# EPICS substitutions: citestApp/Db/user.substitutions
# Example substitutions file

file "db/dbExample1.db" {
    { user = "sdcswd" }
}

file db/dbExample2.db {
    pattern { user, no, scan }
        { "sdcswd", 1, "1 second" }
        { "sdcswd", 2, "2 second" }
        { "sdcswd", 3, "5 second" }
}
